TYPE "Prod_SetUp_Aut_Feedbak"
VERSION : 0.1
// Block: Prod_SetUp_Aut_Feedbak
   STRUCT
      Assi_Profilatrice_InPosizione : Bool;
      Assi_Bordatrice_InPosizione : Bool;
   END_STRUCT;

END_TYPE
